% RSLogix 500 project DDE-Messaging.RSS, saved by version 8.30.00.16 %
PROJECT "UNTITLED"    % processor: Bul.1763 MicroLogix 1100 Series B %

PROGRAM FILES
  LAD 2 "MAIN"  3 rungs
  LAD 3 "TIMER"  10 rungs
  LAD 4 "COUNTER"  5 rungs

DATA FILES
  O0 OUTPUT  4 elements
  I1 INPUT  6 elements
  S2 STATUS  66 elements
  B3 BINARY  1 elements
  T4 TIMER  1 elements
  C5 COUNTER  1 elements
  R6 CONTROL  1 elements
  N7 INTEGER  5 elements
  F8 FLOAT  1 elements
  ST9 STRING  7 elements

LADDER 2 "MAIN"
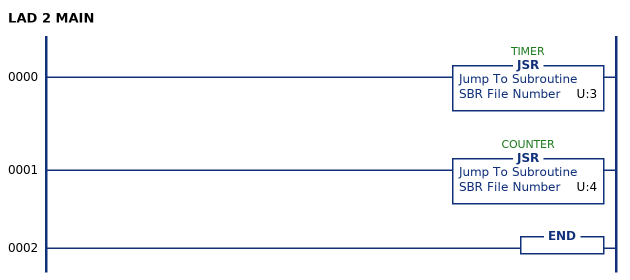
% Rung: 0 %
SOR JSR U:3 EOR
%   U:3  "TIMER" %
% Rung: 1 %
SOR JSR U:4 EOR
%   U:4  "COUNTER" %
% Rung: 2 %
SOR END EOR

LADDER 3 "TIMER"
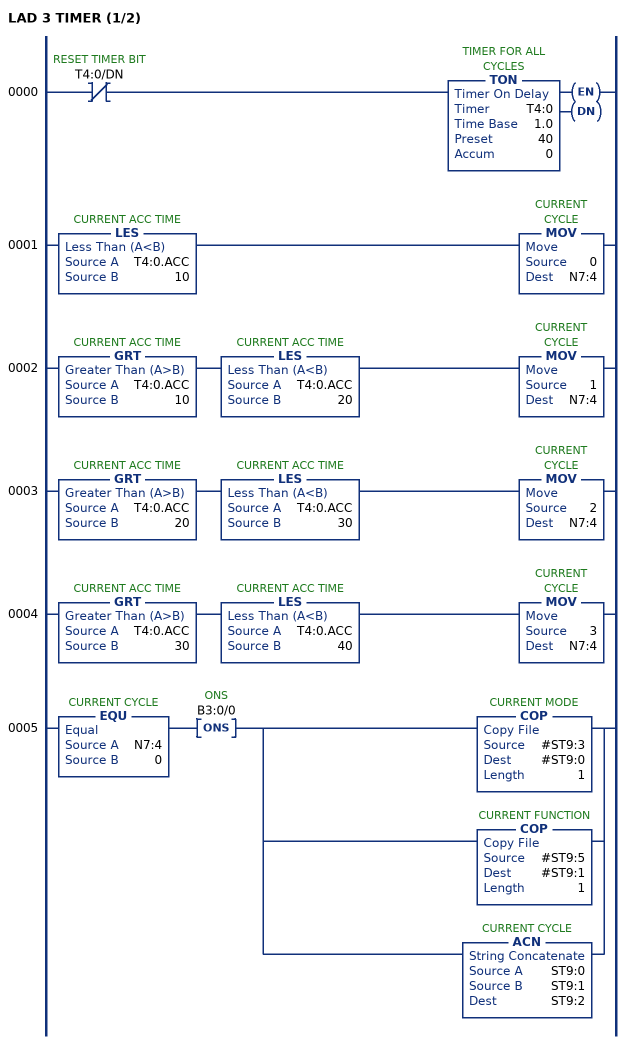
% Rung: 0 %
SOR XIO T4:0/DN TON T4:0 1.0 40 0 EOR
%   T4:0/DN  "RESET TIMER BIT" %
%   T4:0  "TIMER FOR ALL CYCLES" %
% Rung: 1 %
SOR LES T4:0.ACC 10 MOV 0 N7:4 EOR
%   T4:0.ACC  "CURRENT ACC TIME" %
%   N7:4  "CURRENT CYCLE" %
% Rung: 2 %
SOR GRT T4:0.ACC 10 LES T4:0.ACC 20 MOV 1 N7:4 EOR
%   T4:0.ACC  "CURRENT ACC TIME" %
%   N7:4  "CURRENT CYCLE" %
% Rung: 3 %
SOR GRT T4:0.ACC 20 LES T4:0.ACC 30 MOV 2 N7:4 EOR
%   T4:0.ACC  "CURRENT ACC TIME" %
%   N7:4  "CURRENT CYCLE" %
% Rung: 4 %
SOR GRT T4:0.ACC 30 LES T4:0.ACC 40 MOV 3 N7:4 EOR
%   T4:0.ACC  "CURRENT ACC TIME" %
%   N7:4  "CURRENT CYCLE" %
% Rung: 5 %
SOR EQU N7:4 0 ONS B3:0/0 BST COP #ST9:3 #ST9:0 1 NXB BST COP #ST9:5 #ST9:1 1 NXB ACN ST9:0 ST9:1 ST9:2 BND BND EOR
%   N7:4  "CURRENT CYCLE" %
%   B3:0/0  "ONS" %
%   ST9:3  "MODE 1" %
%   ST9:0  "CURRENT MODE" %
%   ST9:5  "FUNCTION1" %
%   ST9:1  "CURRENT FUNCTION" %
%   ST9:2  "CURRENT CYCLE" %

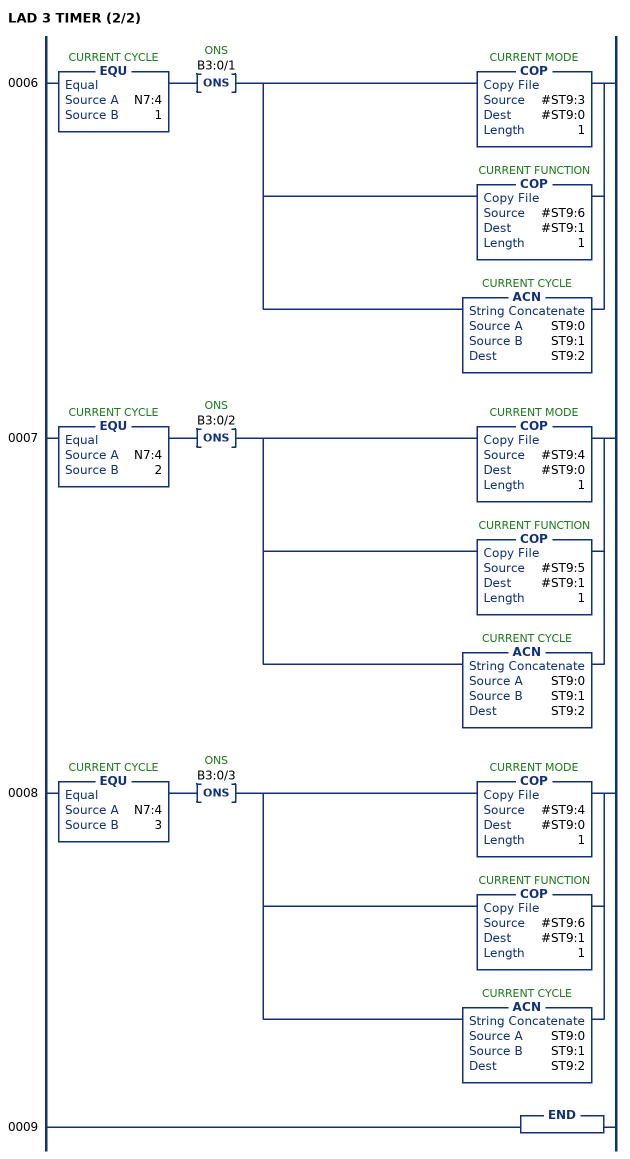
% Rung: 6 %
SOR EQU N7:4 1 ONS B3:0/1 BST COP #ST9:3 #ST9:0 1 NXB BST COP #ST9:6 #ST9:1 1 NXB ACN ST9:0 ST9:1 ST9:2 BND BND EOR
%   N7:4  "CURRENT CYCLE" %
%   B3:0/1  "ONS" %
%   ST9:3  "MODE 1" %
%   ST9:0  "CURRENT MODE" %
%   ST9:6  "FUNCTION2" %
%   ST9:1  "CURRENT FUNCTION" %
%   ST9:2  "CURRENT CYCLE" %
% Rung: 7 %
SOR EQU N7:4 2 ONS B3:0/2 BST COP #ST9:4 #ST9:0 1 NXB BST COP #ST9:5 #ST9:1 1 NXB ACN ST9:0 ST9:1 ST9:2 BND BND EOR
%   N7:4  "CURRENT CYCLE" %
%   B3:0/2  "ONS" %
%   ST9:4  "MODE2" %
%   ST9:0  "CURRENT MODE" %
%   ST9:5  "FUNCTION1" %
%   ST9:1  "CURRENT FUNCTION" %
%   ST9:2  "CURRENT CYCLE" %
% Rung: 8 %
SOR EQU N7:4 3 ONS B3:0/3 BST COP #ST9:4 #ST9:0 1 NXB BST COP #ST9:6 #ST9:1 1 NXB ACN ST9:0 ST9:1 ST9:2 BND BND EOR
%   N7:4  "CURRENT CYCLE" %
%   B3:0/3  "ONS" %
%   ST9:4  "MODE2" %
%   ST9:0  "CURRENT MODE" %
%   ST9:6  "FUNCTION2" %
%   ST9:1  "CURRENT FUNCTION" %
%   ST9:2  "CURRENT CYCLE" %
% Rung: 9 %
SOR END EOR

LADDER 4 "COUNTER"
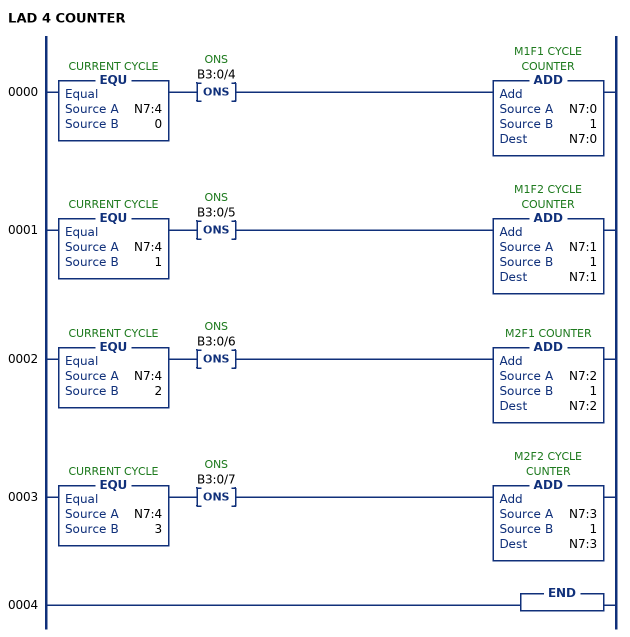
% Rung: 0 %
SOR EQU N7:4 0 ONS B3:0/4 ADD N7:0 1 N7:0 EOR
%   N7:4  "CURRENT CYCLE" %
%   B3:0/4  "ONS" %
%   N7:0  "M1F1 CYCLE COUNTER" %
% Rung: 1 %
SOR EQU N7:4 1 ONS B3:0/5 ADD N7:1 1 N7:1 EOR
%   N7:4  "CURRENT CYCLE" %
%   B3:0/5  "ONS" %
%   N7:1  "M1F2 CYCLE COUNTER" %
% Rung: 2 %
SOR EQU N7:4 2 ONS B3:0/6 ADD N7:2 1 N7:2 EOR
%   N7:4  "CURRENT CYCLE" %
%   B3:0/6  "ONS" %
%   N7:2  "M2F1 COUNTER" %
% Rung: 3 %
SOR EQU N7:4 3 ONS B3:0/7 ADD N7:3 1 N7:3 EOR
%   N7:4  "CURRENT CYCLE" %
%   B3:0/7  "ONS" %
%   N7:3  "M2F2 CYCLE CUNTER" %
% Rung: 4 %
SOR END EOR

OTHER DOCUMENTED ADDRESSES
  PFILE:4  "COUNTER"

DATA TABLE (non-zero values as saved)
DATA T4
% .PRE .ACC %
% T4:0 % 40 0
DATA ST9
% ST9:0 % "M2"
% ST9:1 % "F1"
% ST9:2 % "M2F1"
% ST9:3 % "M1"
% ST9:4 % "M2"
% ST9:5 % "F1"
% ST9:6 % "F2"
